FUNCTION_BLOCK NodeInit (* Template for a Basic Function Block Type *)
  (* Standard: 61499-2 *)
  (* Version 1.0, 2021-07-28, Tuojian Lyu *)
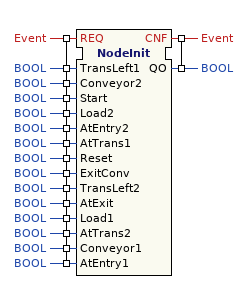
  EVENT_INPUT
    REQ WITH TransLeft1, Conveyor2, Start, Load2, AtEntry2, AtTrans1, Reset, ExitConv, TransLeft2, AtExit, Load1, AtTrans2, Conveyor1, AtEntry1; (* Normal Execution Request *)
  END_EVENT
  EVENT_OUTPUT
    CNF WITH QO; (* Execution Confirmation *)
  END_EVENT
  VAR_INPUT
    TransLeft1 : BOOL; (* Input event qualifier *)
    Conveyor2 : BOOL;
    Start : BOOL;
    Load2 : BOOL;
    AtEntry2 : BOOL;
    AtTrans1 : BOOL;
    Reset : BOOL;
    ExitConv : BOOL;
    TransLeft2 : BOOL;
    AtExit : BOOL;
    Load1 : BOOL;
    AtTrans2 : BOOL;
    Conveyor1 : BOOL;
    AtEntry1 : BOOL;
  END_VAR
  VAR_OUTPUT
    QO : BOOL; (* Output event qualifier *)
  END_VAR
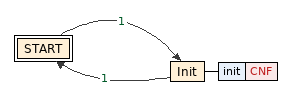
  EC_STATES
    START; (* Initial State *)
    Init : init -> CNF;
  END_STATES
  EC_TRANSITIONS
    START TO Init := 1;
    Init TO START := 1;
  END_TRANSITIONS
  ALGORITHM init IN ST:

  END_ALGORITHM
END_FUNCTION_BLOCK
